TYPE (* a Struct holding 8 Object IDs *)
  (* Version 1.0, 2026-05-28, Franz Höpfinger, Demmler Andreas Fahrzeugbau *)
  PACKAGE isobus::UT::Q::types;
  IMPORT isobus::UT::Q::const::IDs::ID_NULL;
  s8ObjectIDs : STRUCT
    u16ObjId01 : UINT := ID_NULL; (* Object ID 1 *)
    u16ObjId02 : UINT := ID_NULL; (* Object ID 2 *)
    u16ObjId03 : UINT := ID_NULL; (* Object ID 3 *)
    u16ObjId04 : UINT := ID_NULL; (* Object ID 4 *)
    u16ObjId05 : UINT := ID_NULL; (* Object ID 5 *)
    u16ObjId06 : UINT := ID_NULL; (* Object ID 6 *)
    u16ObjId07 : UINT := ID_NULL; (* Object ID 7 *)
    u16ObjId08 : UINT := ID_NULL; (* Object ID 8 *)
  END_STRUCT;
END_TYPE
